FUNCTION_BLOCK FB_System_AKM_Ablaufsteuerung
VAR_IN_OUT
	Zustand			: ST_System_AKM_Zustand;
	Stellwert		: ST_System_AKM_Stellwert;
	Steuerung		: ST_System_AKM_Steuerung;
END_VAR
VAR_INPUT

	Parameter		: ST_System_AKM_Parameter;
END_VAR
VAR_OUTPUT
END_VAR
VAR
	Timer			: TON;
	E_AKM_Zustand_Status_Idle_Sperre		: SINT;
	E_AKM_Zustand_Status_Stoerung		: SINT;
	E_AKM_Zustand_Status_Betriebsbereit 	: SINT;
	E_AKM_Zustand_Status_Nachl			: SINT;
	E_AKM_Zustand_Status_Betrieb			: SINT;
	E_AKM_Zustand_Status_Betrieb_Sperre	: SINT;
	E_AKM_Zustand_Status_Vorl			: SINT;

END_VAR

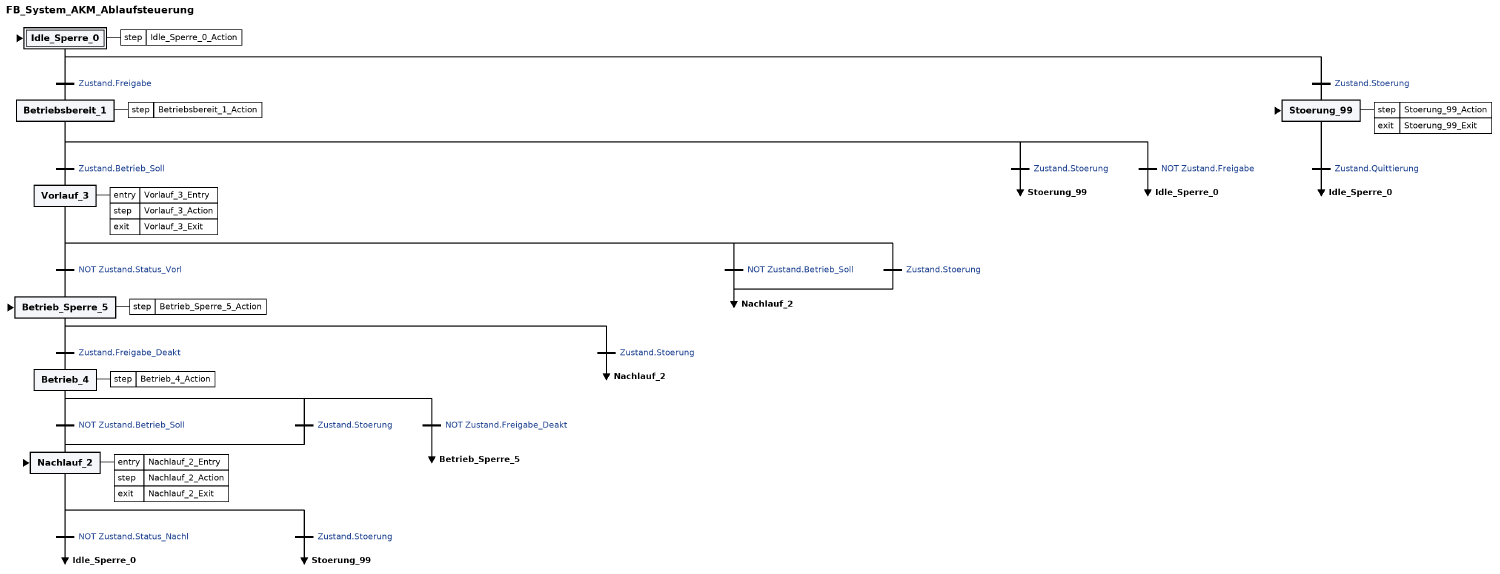
INITIAL_STEP Idle_Sperre_0:
    Idle_Sperre_0_Action(N);  // step action
END_STEP
TRANSITION FROM Idle_Sperre_0 TO Betriebsbereit_1
    := Zustand.Freigabe;
END_TRANSITION
TRANSITION FROM Idle_Sperre_0 TO Stoerung_99
    := Zustand.Stoerung;
END_TRANSITION
STEP Stoerung_99:
    Stoerung_99_Action(N);  // step action
    Stoerung_99_Exit(P0);  // exit action
END_STEP
TRANSITION FROM Stoerung_99 TO Idle_Sperre_0
    := Zustand.Quittierung;
END_TRANSITION
STEP Betriebsbereit_1:
    Betriebsbereit_1_Action(N);  // step action
END_STEP
TRANSITION FROM Betriebsbereit_1 TO Vorlauf_3
    := Zustand.Betrieb_Soll;
END_TRANSITION
TRANSITION FROM Betriebsbereit_1 TO Stoerung_99
    := Zustand.Stoerung;
END_TRANSITION
TRANSITION FROM Betriebsbereit_1 TO Idle_Sperre_0
    := NOT Zustand.Freigabe;
END_TRANSITION
STEP Vorlauf_3:
    Vorlauf_3_Entry(P1);  // entry action
    Vorlauf_3_Action(N);  // step action
    Vorlauf_3_Exit(P0);  // exit action
END_STEP
TRANSITION FROM Vorlauf_3 TO Betrieb_Sperre_5
    := NOT Zustand.Status_Vorl;
END_TRANSITION
TRANSITION FROM Vorlauf_3 TO Nachlauf_2
    := NOT Zustand.Betrieb_Soll;
END_TRANSITION
TRANSITION FROM Vorlauf_3 TO Nachlauf_2
    := Zustand.Stoerung;
END_TRANSITION
STEP Betrieb_Sperre_5:
    Betrieb_Sperre_5_Action(N);  // step action
END_STEP
TRANSITION FROM Betrieb_Sperre_5 TO Betrieb_4
    := Zustand.Freigabe_Deakt;
END_TRANSITION
TRANSITION FROM Betrieb_Sperre_5 TO Nachlauf_2
    := Zustand.Stoerung;
END_TRANSITION
STEP Betrieb_4:
    Betrieb_4_Action(N);  // step action
END_STEP
TRANSITION FROM Betrieb_4 TO Nachlauf_2
    := NOT Zustand.Betrieb_Soll;
END_TRANSITION
TRANSITION FROM Betrieb_4 TO Nachlauf_2
    := Zustand.Stoerung;
END_TRANSITION
TRANSITION FROM Betrieb_4 TO Betrieb_Sperre_5
    := NOT Zustand.Freigabe_Deakt;
END_TRANSITION
STEP Nachlauf_2:
    Nachlauf_2_Entry(P1);  // entry action
    Nachlauf_2_Action(N);  // step action
    Nachlauf_2_Exit(P0);  // exit action
END_STEP
TRANSITION FROM Nachlauf_2 TO Idle_Sperre_0
    := NOT Zustand.Status_Nachl;
END_TRANSITION
TRANSITION FROM Nachlauf_2 TO Stoerung_99
    := Zustand.Stoerung;
END_TRANSITION

ACTION Betrieb_4_Action:
(* Stellwert setzen *)
Stellwert.Betrieb := TRUE;

(* Zustand setzen *)
Zustand.Betrieb	:= TRUE;
Zustand.Status := E_AKM_Zustand_Status_Betrieb;
END_ACTION

ACTION Betrieb_Sperre_5_Action:
(* Stellwert setzen *)
Stellwert.Betrieb := TRUE;

(* Zustand setzen *)
Zustand.Betrieb	:= TRUE;
Zustand.Status := E_AKM_Zustand_Status_Betrieb_Sperre;
END_ACTION

ACTION Betriebsbereit_1_Action:
(* Stellwert setzen *)
Stellwert.Betrieb := FALSE;

(* Zustand setzen *)
Zustand.Betrieb	:= FALSE;
Zustand.Status := E_AKM_Zustand_Status_Betriebsbereit;
END_ACTION

ACTION Idle_Sperre_0_Action:
(* Stellwert setzen *)
Stellwert.Betrieb := FALSE;

(* Zustand setzen *)
Zustand.Betrieb	:= FALSE;
Zustand.Status := E_AKM_Zustand_Status_Idle_Sperre;

(* Quittierungszustand auf False setzen, damit das System bei einer erneuten Störung nicht direkt wieder angeschaltet wird *)
Steuerung.Quittierung	:= FALSE;
END_ACTION

ACTION Nachlauf_2_Action:
(* Nachlauf Timer starten *)
Timer( 	IN := Zustand.Status_Nachl,
		PT := REAL_TO_TIME(Parameter.Zeit_Nachl)
);
Zustand.Status_Nachl	:= NOT(Timer.Q AND NOT Zustand.Betrieb);

(* Stellwert setzen *)
Stellwert.Betrieb := FALSE;

(* Zustand setzen *)
Zustand.Betrieb	:= FALSE;
Zustand.Status := E_AKM_Zustand_Status_Nachl;
END_ACTION

ACTION Nachlauf_2_Entry:
Zustand.Status_Nachl := TRUE;
(* Reset Timer *)
Timer(IN := FALSE);
END_ACTION

ACTION Nachlauf_2_Exit:
Zustand.Status_Nachl := FALSE;
END_ACTION

ACTION Stoerung_99_Action:
(* Stellwert setzen *)
Stellwert.Betrieb := FALSE;

(* Zustand setzen *)
Zustand.Stoerung := TRUE;
Zustand.Betrieb	:= FALSE;
Zustand.Status := E_AKM_Zustand_Status_Stoerung;
END_ACTION

ACTION Stoerung_99_Exit:
Zustand.Stoerung	:= FALSE;
END_ACTION

ACTION Vorlauf_3_Action:
(* Vorlaufzeit Timer starten *)
Timer( 	IN := Zustand.Status_Vorl,
		PT := REAL_TO_TIME(Parameter.Zeit_Vorl)
);
Zustand.Status_Vorl := NOT (Timer.Q AND Zustand.Betrieb);

(* Stellwert setzen *)
Stellwert.Betrieb := TRUE;

(* Zustand setzen *)
Zustand.Betrieb	:= FALSE;
Zustand.Status := E_AKM_Zustand_Status_Vorl;
END_ACTION

ACTION Vorlauf_3_Entry:
Zustand.Status_Vorl := TRUE;
(* Reset Timer *)
Timer(IN := FALSE);
END_ACTION

ACTION Vorlauf_3_Exit:
Zustand.Status_Vorl := FALSE;
END_ACTION

END_FUNCTION_BLOCK

(* stored: Version 1.1.0.1, ProductVersion 3.1.4024.9
   POU FB_System_AKM_Ablaufsteuerung: Id {cb18b568-4110-4f3d-ab1b-878eb521f078}, SpecialFunc None
   Action Betrieb_4_Action: Id {005f679c-41c5-4551-82f3-20211e6856c8}
   Action Betrieb_Sperre_5_Action: Id {9ffc5cac-fda7-4b13-952d-891076123fab}
   Action Betriebsbereit_1_Action: Id {c1e97e4c-a8fd-4220-bf1f-d76c77930c55}
   Action Idle_Sperre_0_Action: Id {03c5badf-9c68-495e-8750-a0809b03c9e9}
   Action Nachlauf_2_Action: Id {ad0ae86d-4a8c-403f-8014-46d52567deb4}
   Action Nachlauf_2_Entry: Id {eaa96422-e9ff-4e36-a4bc-1bba897a878d}
   Action Nachlauf_2_Exit: Id {dbb5973e-1495-4851-bd89-09c9788b1238}
   Action Stoerung_99_Action: Id {08eba25d-fdd0-4c0c-9e45-d8f2df5806df}
   Action Stoerung_99_Exit: Id {59e1a436-fc41-4ca4-a2ab-273de44c967a}
   Action Vorlauf_3_Action: Id {25110893-37b3-43c3-8da1-3def828e035a}
   Action Vorlauf_3_Entry: Id {7a5ca0e6-7f47-48a2-aea9-5b2a915d5724}
   Action Vorlauf_3_Exit: Id {0254ce04-ba7d-44ad-b60f-5b20b69d4378} *)
